// This function has been automatically generated from the project information.
{attribute 'signature_flag' := '1073741824'}
{attribute 'TcGenerated'}
{attribute 'no-analysis'}
FUNCTION F_GetTitle : WSTRING
VAR_INPUT
	
END_VAR

F_GetTitle := "CNM Recipe Handling";

END_FUNCTION

(* stored: Version 1.1.0.1
   POU F_GetTitle: Id {b37f940f-5fe5-4855-8606-7235bee2fed9}, SpecialFunc None *)
